GLOBALCONSTANTS myComputers (* Global constants *)
  (* Standard: 61499-1 *)
  (* Version 1.0, 2023-10-22, franz *)
  VAR_GLOBAL CONSTANT
    C_PC_A : WSTRING := "192.168.178.60:61499";
    C_PC_B : WSTRING := "192.168.178.62:61499";
  END_VAR
END_GLOBALCONSTANTS
